// TIA Portal V17 export
// export: Created 2025-01-08T13:55:36.941715Z, ExportSetting WithDefaults, DisplayName Totally Integrated Automation Portal, DisplayVersion V17, DisplayName TIA Portal Openness, DisplayVersion V17, DisplayName TIA Portal Version Control Interface, DisplayVersion V17, DisplayName SINAMICS Startdrive Advanced, DisplayVersion V17 Update2, DisplayName SINAMICS Startdrive G130, G150, S120, S150, SINAMICS MV, S210, DisplayVersion V17 Update2, DisplayName SINAMICS Startdrive G110M, G120, G120C, G120D, G120P, G115D, DisplayVersion V17 Update2, DisplayName STEP 7 Professional, DisplayVersion V17, DisplayName STEP 7 Safety, DisplayVersion V17, DisplayName WinCC Advanced, DisplayVersion V17
TYPE "HSMMachineParaMask3"
// stored: IsFailsafeCompliant false
   STRUCT
      iSync3OutputDelay : Bool;
      iSync3OutputLenght : Bool;
      iTeachTolerance : Bool;
      iSynch1Mode : Bool;
      iSynch2Mode : Bool;
      iSynch3Mode : Bool;
      iOverCurrentCorrection : Bool;
      iServiceFeedRate : Bool;
      iPreFeedMode : Bool;
      iPreFeed : Bool;
      iLabelSensorWindowPreFeedLenght : Bool;
      iLabelSensorCount : Bool;
      "iSPS-Mode" : Bool;
      iZdtWin : Bool;
      iDistRes : Bool;
      "iSPS-DB-No-Ctrl" : Bool;
   END_STRUCT;
END_TYPE
